{attribute 'GeneratedUsingTerminal: EPP1322-0001-0017'}
{attribute addProperty VendorId "#x00000002"}
{attribute addProperty BoxType "EPP1322-0001-0017"}
{attribute addProperty Description "EPP1322-0001 3 port EtherCAT P gateway"}
{attribute addProperty Physics "YYYY"}
{attribute addProperty Id "InfoDataAT %I*InfoData_6F19DB2B2"}
{attribute addProperty CRC "532711307"}
{attribute addProperty Size "2"}
TYPE EPP1322_1FC0878B EXTENDS TcoIo.EtcSlaveBoxBase_77A0E4A7 :
STRUCT
	{attribute addProperty Name "InfoData"}
	InfoData : TcoIo.InfoData_6F19DB2B;
END_STRUCT
END_TYPE

(* stored: Version 1.2.0.0
   DUT EPP1322_1FC0878B: Id {7221ecdd-10dd-4ff0-b992-88a7b46eefc1} *)
